{attribute 'pack_mode' := '2'}
TYPE ST_FLY_STATE :
STRUCT
  eState              : E_AXIS_STATE; // mirror the requested command + E_PROGRESS
END_STRUCT
END_TYPE

(* stored: Version 1.1.0.1, ProductVersion 3.1.4026.18
   DUT ST_FLY_STATE: Id {cb808a36-4205-4e7f-bb65-56e9c77e1e0e} *)
